FUNCTION MF_Gaussian : real
VAR_INPUT
	x,d,c:REAL;(*Membership function parameters,
specified as the vector [d c], where σ is the 
standard deviation AND c is the mean.*)
END_VAR
VAR_OUTPUT
	Error:BOOL;
END_VAR

IF NOT(d=0) THEN
	MF_Gaussian := LREAL_TO_REAL(EXP(-EXPT((x-c),2)/EXPT(2*d,2)));
ELSE
	Error:=TRUE;
END_IF

END_FUNCTION

(* stored: Version 1.1.0.1, ProductVersion 3.1.4024.6
   POU MF_Gaussian: Id {49d82a09-a965-43d9-8aae-c37daf3c46fb}, SpecialFunc None *)
